{attribute 'linkalways'} 
{attribute 'no_explicit_call' := 'This FB is a CLASS and must be accessed using methods or properties'}
{attribute 'enable_dynamic_creation'}
FUNCTION_BLOCK FINAL ADD_LREAL EXTENDS Node
VAR
	in1 : _LREAL(0.0);
	in2 : _LREAL(0.0);
	out : _LREAL(0.0);
END_VAR

METHOD PUBLIC Clone : I_Node
VAR
	pNode : POINTER TO ADD_LREAL;
END_VAR
pNode := __NEW(ADD_LREAL);
Clone := pNode^;
END_METHOD

METHOD FB_init : BOOL
VAR_INPUT
	bInitRetains : BOOL; // if TRUE, the retain variables are initialized (warm start / cold start)
	bInCopyCode : BOOL;  // if TRUE, the instance afterwards gets moved into the copy code (online change)
END_VAR
AddInput('in1',THIS^.in1);
AddInput('in2',THIS^.in2);
AddOutput('out', THIS^.out);
END_METHOD

METHOD PROTECTED OnExecute
VAR
END_VAR
out.Value := in1.Value + in2.Value;
END_METHOD

END_FUNCTION_BLOCK

(* stored: Version 1.1.0.1, ProductVersion 3.1.4024.15
   POU ADD_LREAL: Id {5b850cfb-c3aa-42d9-bcee-4b1fac4481bc}, SpecialFunc None
   Folder Constructor: Id {e8b19b0c-d482-4b8d-b7f9-61ae1cfbc4d5}
   Method Clone: Id {0f6ae499-4995-479c-bcd8-dfd88ddffde1}
   Method FB_init: Id {55722133-4cb1-4e92-8798-8ade0917644c}
   Method OnExecute: Id {9959b398-77f1-47d1-b877-effdd044b38b} *)
